{attribute 'qualified_only'}
{attribute 'strict'}
{attribute 'to_string'}
TYPE MotorStatus :
(
	Aan := 0,
	Uit
);
END_TYPE

(* stored: Version 1.1.0.1
   DUT MotorStatus: Id {733f9dd0-353e-4e31-926e-9fcc3743effe} *)
